Fanuc KAREL source: kc00031.KL

-- PROVISIONAL review KL for V1013-1; original PC SHA256 049795d1505989b8110ecf01cac4f44bc113d4bbc6a653cea5a1e122bae76bb6
-- Incomplete behavior may be omitted. Consult companion uncertainty JSON. Do not deploy.
PROGRAM KC00031
%NOLOCKGROUP
BEGIN
  -- UNRESOLVED_PC offsets 5-27; opcodes 27,22,22,31,23
  -- UNRESOLVED_PC offsets 32-36; opcodes 7F
END KC00031
